Fanuc TP program (LS listing): UP002.LS

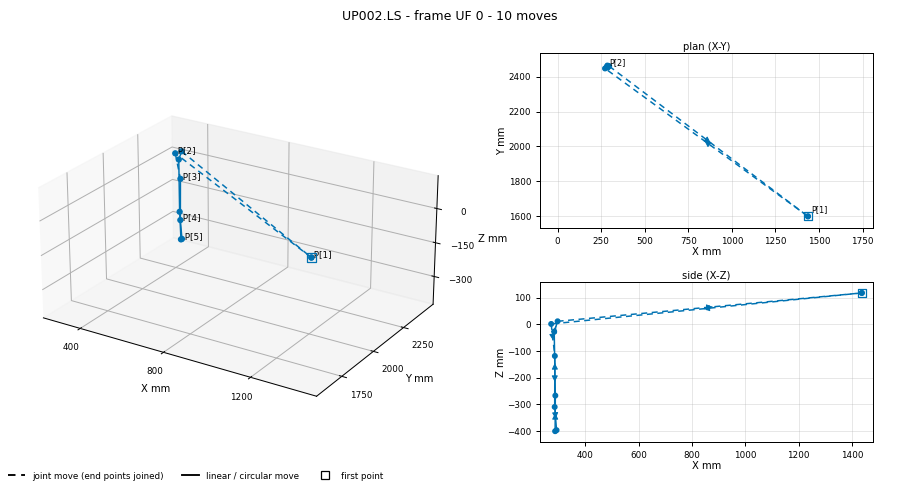
[picture p0: tool path of UP002.LS in frame UF 0, 10 of 10 moves have a stored position in this frame; points joined in program order, loops and branches not executed]
/PROG  UP002
/ATTR
OWNER		= MNEDITOR;
COMMENT		= "TOMA ST1140-1 ";
PROG_SIZE	= 5460;
CREATE		= DATE 23-12-14  TIME 14:23:16;
MODIFIED	= DATE 24-05-06  TIME 18:42:16;
FILE_NAME	= UP022;
VERSION		= 0;
LINE_COUNT	= 25;
MEMORY_SIZE	= 9336;
PROTECT		= READ_WRITE;
TCD:  STACK_SIZE	= 500,
      TASK_PRIORITY	= 50,
      TIME_SLICE	= 0,
      BUSY_LAMP_OFF	= 0,
      ABORT_REQUEST	= 0,
      PAUSE_REQUEST	= 0;
DEFAULT_GROUP	= 1,1,1,1,*;
CONTROL_CODE	= 00000000 00000000;
/APPL
/MN
   1:  UFRAME_NUM=0 ;
   2:  UTOOL_NUM=2 ;
   3:  PAYLOAD[2] ;
   4:  !Apagar Perfil Lib 77 vs ST1140-1 ;
   5:J P[1] 100% CNT0 ACC100 TB    .10sec,P-SPS    ;
      1:  TC_ONLINE (ON) ;
      2:  DO[23]=OFF ;
      3:  TIMER[4]=RESET ;
      4:  TIMER[4]=START ;
      5:  CALL MAKRO050    ;
      6:  !Lib. de Herramientas ;
      7:  DO[80]=ON ;
      8:  DO[78]=OFF ;
      9:  DO[77]=ON ;
     10:  DO[75]=OFF ;
     11:  DO[74]=ON ;
     12:  DO[73]=ON ;
     13:  DO[71]=OFF ;
     14:  DO[70]=OFF ;
     15:  DO[69]=OFF ;
     16:  DO[68]=OFF ;
     17:  DO[67]=OFF ;
     18:  !Lib. de Anticolisiones ;
     19:  DO[41]=ON ;
     20:  DO[42]=ON ;
     21:  DO[43]=ON ;
     22:  DO[44]=ON ;
     23:  DO[45]=ON ;
     24:  DO[46]=ON ;
     25:  !Apagar Posicion Base ;
     26:  DO[15]=OFF ;
     27:  !Robot en Trayectoria ;
     28:   ;
     29:  F[4]=(ON) ;
     30:  CALL MAKRO343    ;
     31:  WAIT (M[38])    ;
     32:  DO[16]=ON ;
     33:  WAIT (M[3] AND M[27] AND DI[77] AND DI[64] AND !DI[63])    ;
     34:  DO[77]=OFF ;
     35:  WAIT (DI[23])    ;
     36:  DO[23]=ON ;
     37:  !Marcas de Usuario: ;
     38:  !Marca 5 Estado de Garra ;
     39:  !Valvula 1 en V, 2-7 en R ;
     40:  !M[21]=(M[32] AND M[35] AND M[37] ;
     41:  !AND M[39] AND M[41] AND M[43]) ;
     42:  TC_ONLINE (!DI[63] AND DI[64] AND DI[77] AND M[3] AND M[27] AND M[30] AND M[95] AND M[96]) ;
       ------ ;
   6:J P[2] 100% CNT100 ACC100 TB   0.00sec,P-SPS    ;
      1:  TC_ONLINE (!DI[63] AND DI[64] AND DI[77] AND M[3] AND M[27] AND M[30] AND M[95] AND M[96]) ;
       ------ ;
   7:J P[3] 100% CNT100 ACC100 TB   0.00sec,P-SPS    ;
      1:  TC_ONLINE (!DI[63] AND DI[64] AND DI[77] AND M[27] AND M[30] AND M[95] AND M[96]) ;
       ------ ;
   8:L P[4] 100mm/sec CNT0 ACC100 TB    .10sec,P-SPS    ;
      1:  TC_ONLINE (!DI[63] AND DI[64] AND DI[77] AND M[27] AND M[30] AND M[95] AND M[96]) ;
       ------ ;
   9:L P[5] 100mm/sec CNT0 ACC100 TB    .10sec,P-SPS    ;
      1:  TC_ONLINE (!DI[63] AND DI[64] AND DI[77] AND M[27] AND M[30] AND M[95] AND M[96]) ;
       ------ ;
  10:   ;
  11:  !En Posicion ST1140-1 ;
  12:  !Tomar Piezas en ST1140-1 ;
  13:  !Fin de Trabajo 2 ;
  14:L P[6] 100mm/sec CNT0 ACC100 TB    .10sec,P-SPS    ;
      1:  TC_ONLINE (ON) ;
      2:  DO[23]=OFF ;
      3:  WAIT (M[1])    ;
      4:  F[5]=(ON) ;
      5:  IF (!DI[15]),F[17]=(ON) ;
      6:  CALL MAKRO343    ;
      7:  WAIT (M[40] AND M[63])    ;
      8:  F[4]=(ON) ;
      9:  CALL MAKRO342    ;
     10:  WAIT (M[37])    ;
     11:   ;
     12:  DO[75]=ON ;
     13:  CALL MAKRO002    ;
     14:  WAIT (DI[76])    ;
     15:  DO[75]=OFF ;
     16:  WAIT (DI[23])    ;
     17:  DO[23]=ON ;
     18:  !Marca 6 Estado de Garra ;
     19:  !Valvula 1,2&5 en V, 3,4,6&7 en R ;
     20:  !M[22]=(M[32] AND M[35] AND M[37] ;
     21:  !AND M[40] AND M[41] AND M[43] ;
     22:  !AND M[63]) ;
     23:  TC_ONLINE (DI[76] AND M[1] AND M[28] AND M[30] AND M[95] AND M[96]) ;
       ------ ;
  15:   ;
  16:L P[7] 300mm/sec CNT0 ACC100 TB    .10sec,P-SPS    ;
      1:  TC_ONLINE (DI[76] AND M[1] AND M[28] AND M[30] AND M[95] AND M[96]) ;
       ------ ;
  17:   ;
  18:  PAYLOAD[2] ;
  19:L P[8] 300mm/sec CNT0 ACC100 TB    .10sec,P-SPS    ;
      1:  TC_ONLINE (DI[76] AND M[1] AND M[28] AND M[30] AND M[95] AND M[96]) ;
       ------ ;
  20:   ;
  21:  !Tomar Piezas CLOSE CLMP3 ;
  22:L P[9] 300mm/sec CNT0 ACC100 TB    .10sec,P-SPS    ;
      1:  TC_ONLINE (ON) ;
      2:  DO[23]=OFF ;
      3:  F[3]=(ON) ;
      4:  CALL MAKRO343    ;
      5:  WAIT (M[36])    ;
      6:  WAIT (DI[63] AND !DI[64])    ;
      7:  WAIT (DI[23])    ;
      8:  DO[23]=ON ;
      9:  !Marca 7 Estado de Garra ;
     10:  !Valvula 1,2,3&5 en V, 4,6&7 en R ;
     11:  !M[23]=(M[32] AND M[36] AND M[37] ;
     12:  !AND M[40] AND M[41] AND M[43] ;
     13:  !AND M[63]) ;
     14:  TC_ONLINE (DI[63] AND !DI[64] AND DI[76] AND M[1] AND M[23] AND M[30] AND M[95] AND M[96]) ;
       ------ ;
  23:   ;
  24:  !Encender Perf Lib 77 vs ST1140-1 ;
  25:J P[10] 100% CNT0 ACC100 TB    .10sec,P-SPS    ;
      1:  TC_ONLINE (ON) ;
      2:  DO[23]=OFF ;
      3:  F[930]=(OFF) ;
      4:  TIMER[4]=STOP ;
      5:  DO[77]=ON ;
      6:  WAIT (DI[23])    ;
      7:  DO[23]=ON ;
      8:  TC_ONLINE (M[1] AND M[23] AND M[30] AND M[95] AND M[96]) ;
       ------ ;
/POS
P[1]{
   GP1:
	UF : 0, UT : 2,		CONFIG : 'N U T, 0, 0, 0',
	X =  1436.857  mm,	Y =  1598.998  mm,	Z =   117.965  mm,
	W =   179.395 deg,	P =    81.558 deg,	R =   -18.495 deg
   GP2:
	UF : 0, UT : 2,
	J1=   100.000  mm
   GP3:
	UF : 0, UT : 2,
	J1=     0.000  mm
   GP4:
	UF : 0, UT : 2,
	J1=     0.000  mm
};
P[2]{
   GP1:
	UF : 0, UT : 2,		CONFIG : 'N U T, 0, 0, 0',
	X =   271.857  mm,	Y =  2447.987  mm,	Z =     1.651  mm,
	W =   -90.741 deg,	P =    84.537 deg,	R =    86.878 deg
   GP2:
	UF : 0, UT : 2,
	J1=   100.000  mm
   GP3:
	UF : 0, UT : 2,
	J1=     0.000  mm
   GP4:
	UF : 0, UT : 2,
	J1=     0.000  mm
};
P[3]{
   GP1:
	UF : 0, UT : 2,		CONFIG : 'N U T, 0, 0, 0',
	X =   285.595  mm,	Y =  2464.811  mm,	Z =  -118.429  mm,
	W =   -86.228 deg,	P =    84.542 deg,	R =    90.277 deg
   GP2:
	UF : 0, UT : 2,
	J1=    98.800  mm
   GP3:
	UF : 0, UT : 2,
	J1=     0.000  mm
   GP4:
	UF : 0, UT : 2,
	J1=     0.000  mm
};
P[4]{
   GP1:
	UF : 0, UT : 2,		CONFIG : 'N U T, 0, 0, 0',
	X =   284.986  mm,	Y =  2461.238  mm,	Z =  -309.592  mm,
	W =   -78.870 deg,	P =    83.508 deg,	R =    95.510 deg
   GP2:
	UF : 0, UT : 2,
	J1=   119.300  mm
   GP3:
	UF : 0, UT : 2,
	J1=     0.000  mm
   GP4:
	UF : 0, UT : 2,
	J1=     0.000  mm
};
P[5]{
   GP1:
	UF : 0, UT : 2,		CONFIG : 'N U T, 0, 0, 0',
	X =   292.052  mm,	Y =  2461.238  mm,	Z =  -396.759  mm,
	W =   -76.141 deg,	P =    85.649 deg,	R =    98.227 deg
   GP2:
	UF : 0, UT : 2,
	J1=   119.301  mm
   GP3:
	UF : 0, UT : 2,
	J1=     0.000  mm
   GP4:
	UF : 0, UT : 2,
	J1=     0.000  mm
};
P[6]{
   GP1:
	UF : 0, UT : 2,		CONFIG : 'N U T, 0, 0, 0',
	X =   286.666  mm,	Y =  2461.866  mm,	Z =  -400.531  mm,
	W =   -82.687 deg,	P =    86.096 deg,	R =    94.960 deg
   GP2:
	UF : 0, UT : 2,
	J1=   120.801  mm
   GP3:
	UF : 0, UT : 2,
	J1=     0.000  mm
   GP4:
	UF : 0, UT : 2,
	J1=     0.000  mm
};
P[7]{
   GP1:
	UF : 0, UT : 2,		CONFIG : 'N U T, 0, 0, 0',
	X =   287.453  mm,	Y =  2452.788  mm,	Z =  -267.032  mm,
	W =   -81.184 deg,	P =    86.096 deg,	R =    94.958 deg
   GP2:
	UF : 0, UT : 2,
	J1=   120.801  mm
   GP3:
	UF : 0, UT : 2,
	J1=     0.000  mm
   GP4:
	UF : 0, UT : 2,
	J1=     0.000  mm
};
P[8]{
   GP1:
	UF : 0, UT : 2,		CONFIG : 'N U T, 0, 0, 0',
	X =   283.253  mm,	Y =  2457.109  mm,	Z =   -27.496  mm,
	W =   -71.710 deg,	P =    84.230 deg,	R =   105.805 deg
   GP2:
	UF : 0, UT : 2,
	J1=   107.400  mm
   GP3:
	UF : 0, UT : 2,
	J1=     0.000  mm
   GP4:
	UF : 0, UT : 2,
	J1=     0.000  mm
};
P[9]{
   GP1:
	UF : 0, UT : 2,		CONFIG : 'N U T, 0, 0, 0',
	X =   295.974  mm,	Y =  2460.949  mm,	Z =    11.625  mm,
	W =   -71.710 deg,	P =    84.230 deg,	R =   105.804 deg
   GP2:
	UF : 0, UT : 2,
	J1=   107.400  mm
   GP3:
	UF : 0, UT : 2,
	J1=     0.000  mm
   GP4:
	UF : 0, UT : 2,
	J1=     0.000  mm
};
P[10]{
   GP1:
	UF : 0, UT : 2,		CONFIG : 'N U T, 0, 0, 0',
	X =  1436.857  mm,	Y =  1598.998  mm,	Z =   117.965  mm,
	W =   179.395 deg,	P =    81.558 deg,	R =   -18.495 deg
   GP2:
	UF : 0, UT : 2,
	J1=   100.000  mm
   GP3:
	UF : 0, UT : 2,
	J1=     0.000  mm
   GP4:
	UF : 0, UT : 2,
	J1=     0.000  mm
};
/END
